PROGRAM INTERNAL FsP_ErrorHandlingPlayground
VAR
	bStart, bDestroy : BOOL;
	pObj, pObj2 : POINTER TO FsFB_ErrorDefinition;
	fbNoError : FsFB_Error;
	fbErrDef : FsFB_ErrorDefinitionOnInit(11, 'Dogs');
	MemArea : FsT_MemArea;
	ipUnk : FsI_Unknown;
	ipObj : FsI_Object;
	pItfs : POINTER TO ARRAY[0..6] OF FsT_Ptr;
	nData, nData2 : FsT_Size;
	sdata : FsT_LStr;
	TaskInfo : FsT_PlcTaskInfo;
END_VAR

fbNoError := fbErrDef;
sData := fbNoError.Message;
fbNoError := FsF_ErrorPath(11,'Cats', ipObj);
sdata := FsF_Error(11,'Cats').Message;
ipUnk := fbNoError;
ipObj := fbNoError;
pItfs := ADR(ipUnk);
pObj2 := ADR(fbNoError);
nData := SIZEOF(fbNoError);
nData2 := FsF_GetSize(ipObj);
TaskInfo :=  FsF_GetPlcTaskInformation();
IF bStart THEN 
	bStart := FALSE;
	pObj := __NEW(FsFB_ErrorDefinition);
	sData := pObj^.TypeName;
	END_IF
IF bDestroy THEN
	bDestroy := FALSE; 
	__DELETE(pObj);
	END_IF

END_PROGRAM

(* stored: Version 1.1.0.1, ProductVersion 3.1.4024.4
   POU FsP_ErrorHandlingPlayground: Id {5a0d939f-a70c-4b2c-82d3-074370e7b7e9}, SpecialFunc None *)
